// TIA Portal V21 export
VAR_GLOBAL   // PLC tag table "K_Motore"
END_VAR
VAR_GLOBAL CONSTANT   // user constants
   K_Motore_AgitatoreVascaProdotto : Int := 1;
   K_Motore_PompaMono : Int := 2;
   K_Motore_CentrifugaLavaggio : Int := 3;
   K_Motore_PompaPistoni : Int := 4;
   K_Motore_PompaOlio : Int := 5;
   K_Motore_PompaRicircoloAcquaCalda : Int := 6;
   K_Motore_PompaRilancioTorre : Int := 7;
   K_Motore_AspiratorePompaPistoni : Int := 8;
END_VAR
